// TIA Portal V20 export
// export: Created 2026-04-18T06:33:56.6156724Z, ExportSetting WithDefaults, DisplayName Totally Integrated Automation Portal, DisplayVersion V20, DisplayName TIA Portal Openness, DisplayVersion V20, DisplayName TIA Portal Version Control Interface, DisplayVersion V20, DisplayName STEP 7 Professional, DisplayVersion V20, DisplayName STEP 7 Safety, DisplayVersion V20, DisplayName WinCC Basic/Comfort/Advanced, DisplayVersion V20
TYPE "UDT_AlarmLimits"
// ============================================================
//  BlockParam Demo - Process Plant Structure
//  Author: Tobias Laubscher
//  Target: TIA Portal V17+
// 
//  Import as external source (SCL). Types compile in order:
//    UDT_AlarmLimits -> UDT_ControlValve -> UDT_EquipmentModule
//    -> UDT_ProcessUnit -> DB_ProcessPlant_A1
// 
//  Hierarchy depth from DB root to leaf:
//    DB -> units[] -> modules[] -> valves[] -> *Limits -> hiLimit  (5 levels)
// 
//  Scale:
//    2 Units x 3 Modules x 4 Valves = 24 Valves
//    24 Valves x 2 Limit blocks      = 48 Alarm blocks
//    48 Alarm blocks x 4 limits      = 192 limit members
//  ============================================================
// stored: IsFailsafeCompliant false
   STRUCT
      hiHiLimit : Real := 100.0;
      hiLimit : Real := 90.0;
      loLimit : Real := 10.0;
      loLoLimit : Real := 5.0;
      hysteresis : Real := 0.5;
      alarmDelay : Time := T#3S;
      enable : Bool := TRUE;
   END_STRUCT;
END_TYPE
